PROGRAM MaintenanceTask
VAR
	CycleCounter: INT := 0;;
	MaintenanceNeeded: BOOL;
	Tclean: Ton;
	
	ResetCounter: BOOL;
	CoffeeReadyOld: BOOL := FALSE;
	
	bResult: BOOL;
	Treset: Ton;
END_VAR

// every cooffee made the counter increase
IF (GVL.CoffeeReady = TRUE) AND (CoffeeReadyOld = FALSE) THEN
    CycleCounter := CycleCounter + 1;
END_IF;

CoffeeReadyOld := GVL.CoffeeReady;

// if the machine has done 5 coffee, the cleaning part is needed
IF CycleCounter >= 5 THEN
    MaintenanceNeeded := TRUE;
   

    Tclean(IN := TRUE, PT := T#6S);
	LogMessage (msg := 'Maintenance required!', cleaning := TRUE);
    IF Tclean.Q THEN
        Tclean(IN := FALSE);
        ResetCounter := TRUE;
		LogMessage(msg := 'Maintenance done', cleaning := FALSE);
    END_IF;
//maintenance finished and numbur of coffe made
ELSE 
    MaintenanceNeeded := FALSE;
    LogMessage(msg := CONCAT('Coffees made: ', INT_TO_STRING(CycleCounter)), cleaning := FALSE);
	;
END_IF;

//after cleaning, counter must be resetted
IF ResetCounter = TRUE THEN  
    
LogMessage(msg := 'Maintenance done', cleaning := FALSE);
Treset(IN := TRUE, PT := T#2S);
    IF Treset.Q THEN
        Treset(IN := FALSE);
		CycleCounter := 0;
        ResetCounter := FALSE;
    END_IF;
END_IF;

END_PROGRAM

(* stored: Version 1.1.0.1, ProductVersion 3.1.4024.15
   POU MaintenanceTask: Id {f2ccf1d7-5961-4f5a-bde9-3b71431e1174}, SpecialFunc None *)
